// TIA Portal V16 export
// export: Created 2022-11-17T11:55:16.9190017Z, ExportSetting WithDefaults, DisplayName Totally Integrated Automation Portal, DisplayVersion V16 Update 6, DisplayName TIA Portal Version Control Interface, DisplayVersion V16 Update 2, DisplayName TIA Portal Openness, DisplayVersion V16 Update 6, DisplayName SINAMICS Startdrive Advanced, DisplayVersion V16 Update 5, DisplayName SINAMICS Startdrive G130, G150, S120, S150, SINAMICS MV, S210, DisplayVersion V16 Update 5, DisplayName SINAMICS Startdrive G110M, G120, G120C, G120D, G120P, G115D, DisplayVersion V16 Update 5, DisplayName STEP 7 Professional, DisplayVersion V16 Update 6, DisplayName STEP 7 Safety, DisplayVersion V16, DisplayName WinCC Advanced, DisplayVersion V16 Update 6
FUNCTION "FC63_StretchPGSAoutPWM" : Void   // FC63, LAD
{ S7_Optimized_Access := 'FALSE' }
AUTHOR : PaZan
VERSION : 0.1
// stored: AutoNumber false, IsIECCheckEnabled false, SetENOAutomatically false, UDAEnableTagReadback false
   VAR_TEMP   // added for the SCL form of the ladder/FBD networks
      _w1 : Bool;
   END_VAR
BEGIN

REGION Network 1
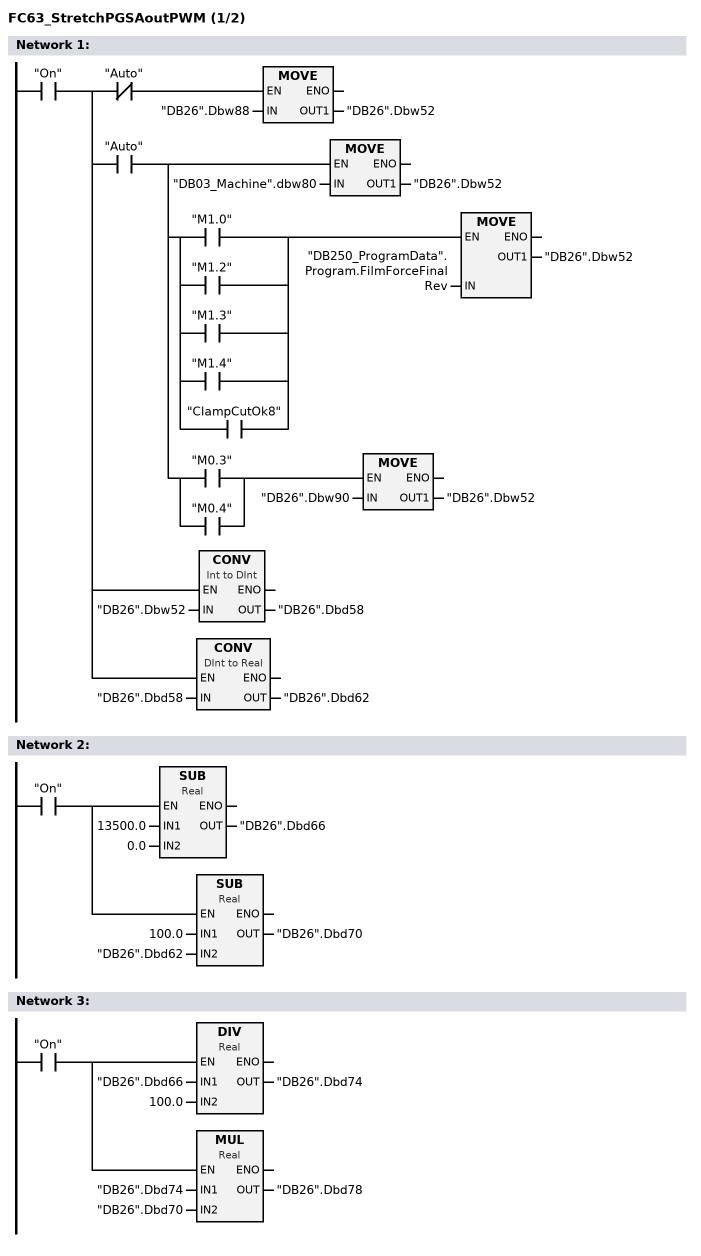
   RUNG wire#powerrail
      Contact( "On" )
      wire#w1
      I_Contact( "Auto" )
      { S7_GenerateENO := "TRUE" } Move(in := "DB26".Dbw88, out1 => "DB26".Dbw52)
   END_RUNG
   RUNG wire#w1
      Contact( "Auto" )
      wire#w2
      { S7_GenerateENO := "TRUE" } Move(in := "DB03_Machine".dbw80, out1 => "DB26".Dbw52)
   END_RUNG
   RUNG wire#w2
      Contact( "M1.0" )
      wire#w3
      { S7_GenerateENO := "TRUE" } Move(in := "DB250_ProgramData".Program.FilmForceFinalRev, out1 => "DB26".Dbw52)
   END_RUNG
   RUNG wire#w2
      Contact( "M1.2" )
   END_RUNG wire#w3
   RUNG wire#w2
      Contact( "M1.3" )
   END_RUNG wire#w3
   RUNG wire#w2
      Contact( "M1.4" )
   END_RUNG wire#w3
   RUNG wire#w2
      Contact( "ClampCutOk8" )
   END_RUNG wire#w3
   RUNG wire#w2
      Contact( "M0.3" )
      wire#w4
      { S7_GenerateENO := "TRUE" } Move(in := "DB26".Dbw90, out1 => "DB26".Dbw52)
   END_RUNG
   RUNG wire#w2
      Contact( "M0.4" )
   END_RUNG wire#w4
   RUNG wire#w1
      { S7_Templates := "[SrcType := Int, DestType := DInt]"; S7_GenerateENO := "TRUE" } Convert(in := "DB26".Dbw52, out => "DB26".Dbd58)
   END_RUNG
   RUNG wire#w1
      { S7_Templates := "[SrcType := DInt, DestType := Real]"; S7_GenerateENO := "TRUE" } Convert(in := "DB26".Dbd58, out => "DB26".Dbd62)
   END_RUNG
   // the same network as SCL:
   IF "On" AND NOT "Auto" THEN "DB26".Dbw52 := "DB26".Dbw88; END_IF;
   #_w1 := "On" AND "Auto";
   IF #_w1 THEN "DB26".Dbw52 := "DB03_Machine".dbw80; END_IF;
   IF #_w1 AND ("M1.0" OR "M1.2" OR "M1.3" OR "M1.4" OR "ClampCutOk8") THEN
       "DB26".Dbw52 := "DB250_ProgramData".Program.FilmForceFinalRev;
   END_IF;
   IF #_w1 AND ("M0.3" OR "M0.4") THEN "DB26".Dbw52 := "DB26".Dbw90; END_IF;
   IF "On" THEN
       "DB26".Dbd58 := INT_TO_DINT("DB26".Dbw52);
       "DB26".Dbd62 := DINT_TO_REAL("DB26".Dbd58);
   END_IF;
END_REGION

REGION Network 2
   RUNG wire#powerrail
      Contact( "On" )
      wire#w1
      { S7_Templates := "SrcType := Real"; S7_GenerateENO := "TRUE" } Sub(in1 := 13500.0, in2 := 0.0, out => "DB26".Dbd66)
   END_RUNG
   RUNG wire#w1
      { S7_Templates := "SrcType := Real"; S7_GenerateENO := "TRUE" } Sub(in1 := 100.0, in2 := "DB26".Dbd62, out => "DB26".Dbd70)
   END_RUNG
   // the same network as SCL:
   IF "On" THEN
       "DB26".Dbd66 := 13500.0 - 0.0;
       "DB26".Dbd70 := 100.0 - "DB26".Dbd62;
   END_IF;
END_REGION

REGION Network 3
   RUNG wire#powerrail
      Contact( "On" )
      wire#w1
      { S7_Templates := "SrcType := Real"; S7_GenerateENO := "TRUE" } Div(in1 := "DB26".Dbd66, in2 := 100.0, out => "DB26".Dbd74)
   END_RUNG
   RUNG wire#w1
      { S7_Templates := "SrcType := Real"; S7_GenerateENO := "TRUE" } Mul(in1 := "DB26".Dbd74, in2 := "DB26".Dbd70, out => "DB26".Dbd78)
   END_RUNG
   // the same network as SCL:
   IF "On" THEN
       "DB26".Dbd74 := "DB26".Dbd66 / 100.0;
       "DB26".Dbd78 := "DB26".Dbd74 * "DB26".Dbd70;
   END_IF;
END_REGION

REGION Network 4: Trunc and copy value for stretch torque in analogic out
   // PAW130
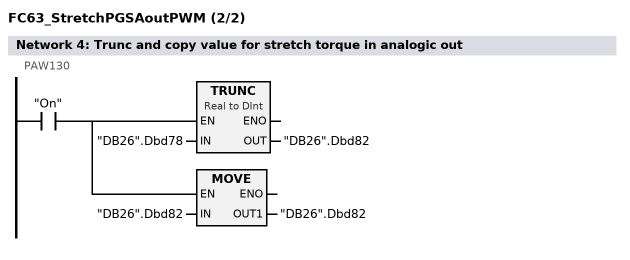
   RUNG wire#powerrail
      Contact( "On" )
      wire#w1
      { S7_Templates := "[SrcType := Real, DestType := DInt]"; S7_GenerateENO := "TRUE" } Trunc(in := "DB26".Dbd78, out => "DB26".Dbd82)
   END_RUNG
   RUNG wire#w1
      { S7_GenerateENO := "TRUE" } Move(in := "DB26".Dbd82, out1 => "DB26".Dbd82)
   END_RUNG
   // the same network as SCL:
   IF "On" THEN
       "DB26".Dbd82 := TRUNC("DB26".Dbd78);
       "DB26".Dbd82 := "DB26".Dbd82;
   END_IF;
END_REGION
END_FUNCTION
